{attribute 'qualified_only'}
{attribute 'strict'}
{attribute 'to_string'}
TYPE HomingMode :
(
	Default := TO_INT(Tc2_Mc2.MC_DefaultHoming),
	Direct := TO_INT(Tc2_Mc2.MC_Direct),
	ForceCalibration := TO_INT(Tc2_Mc2.MC_ForceCalibration),
	ResetCalibration := TO_INT(Tc2_Mc2.MC_ResetCalibration)
);
END_TYPE

(* stored: Version 1.1.0.1
   DUT HomingMode: Id {074f448e-f9f8-4680-b3e7-1573186979b1} *)
